(* CoDeSys 2.3.9.41 project: PLC1.pro *)
(* Libraries: Util.lib 18.5.10 15:14:28, STANDARD.LIB 4.10.05 11:14:46, IECSFC.LIB 13.4.06 15:51:28, SYSLIBTIME.LIB 6.11.19 15:29:28, ANALYZATION.LIB 5.10.99 09:05:06 *)

(* PLC configuration (modules and I/O channels)
Fast discrete inputs [I_SIMPLE_INPUT] node 0, in %IB0 out %QB0 {ChannellName = Fast discrete inputs; Filtrationtime = 10000}
  AT %IX0.0 [BitInput] Discrete input 1 {ChannellName = Enter name}
  AT %IX0.1 [BitInput] Discrete input 2 {ChannellName = Enter name}
  AT %IX0.2 [BitInput] Discrete input 3 {ChannellName = Enter name}
  AT %IX0.3 [BitInput] Discrete input 4 {ChannellName = Enter name}
Discrete inputs [ID130] node 1, in %IB1 out %QB1 {ChannellName = Discrete inputs; Filtrationtime_GeneralINP = 10; PinCount = 12; Visibility = No}
  AT %IB1.0 [ByteInput] 8 discrete inputs {ChannellName = Enter name}
  AT %IB1.1 [ByteInput] 4 discrete inputs {ChannellName = Enter name}
DO1 AT %QX2.0 [BitOutput] Fast discrete output 1 {ChannellName = Enter name}
AT %QX2.1 [BitOutput] Fast discrete output 2 {ChannellName = Enter name}
AT %QX2.2 [BitOutput] Fast discrete output 3 {ChannellName = Enter name}
AT %QX2.3 [BitOutput] Fast discrete output 4 {ChannellName = Enter name}
Discrete outputs [ID131] node 3, in %IB3 out %QB3 {ChannellName = Discrete outputs; SafeValueByte = 0; Visibility = No}
  AT %QB3.0 [ByteOutput] 8 discrete outputs {ChannellName = Enter name}
  AT %QB3.1 [ByteOutput] 8 discrete outputs {ChannellName = Enter name}
Fast analog inputs [ID125] node 4, in %IB4 out %QB4 {ChannellName = Fast analog inputs; Flt_Comm = 50Hz 2Por}
  AT %IR4.0 [FloatInputP] You need to reboot PLC after change AI configuration! {ChannellName = Fast analog input; AIN_TYPE = 4-20 mA; Peak_Filtr = 200; Flt_Ch = Off; TauRC = 10; MinFV = 0; MaxFV = 20000.0}
  AT %IR4.1 [FloatInputP] You need to reboot PLC after change AI configuration! {ChannellName = Fast analog input; AIN_TYPE = 4-20 mA; Peak_Filtr = 200; Flt_Ch = Off; TauRC = 10; MinFV = 0; MaxFV = 20000.0}
  AT %IR4.2 [FloatInputP] You need to reboot PLC after change AI configuration! {ChannellName = Fast analog input; AIN_TYPE = 4-20 mA; Peak_Filtr = 200; Flt_Ch = Off; TauRC = 10; MinFV = 0; MaxFV = 20000.0}
  AT %IR4.3 [FloatInputP] You need to reboot PLC after change AI configuration! {ChannellName = Fast analog input; AIN_TYPE = 4-20 mA; Peak_Filtr = 200; Flt_Ch = Off; TauRC = 10; MinFV = 0; MaxFV = 20000.0}
  AT %IR4.4 [FloatInputP] You need to reboot PLC after change AI configuration! {ChannellName = Fast analog input; AIN_TYPE = 4-20 mA; Peak_Filtr = 200; Flt_Ch = Off; TauRC = 10; MinFV = 0; MaxFV = 20000.0}
  AT %IR4.5 [FloatInputP] You need to reboot PLC after change AI configuration! {ChannellName = Fast analog input; AIN_TYPE = 4-20 mA; Peak_Filtr = 200; Flt_Ch = Off; TauRC = 10; MinFV = 0; MaxFV = 20000.0}
  AT %IR4.6 [FloatInputP] You need to reboot PLC after change AI configuration! {ChannellName = Fast analog input; AIN_TYPE = 4-20 mA; Peak_Filtr = 200; Flt_Ch = Off; TauRC = 10; MinFV = 0; MaxFV = 20000.0}
  AT %IR4.7 [FloatInputP] You need to reboot PLC after change AI configuration! {ChannellName = Fast analog input; AIN_TYPE = 4-20 mA; Peak_Filtr = 200; Flt_Ch = Off; TauRC = 10; MinFV = 0; MaxFV = 20000.0}
  AT %IW4.8 [WordInput] AI read time (10ms) {ChannellName = Enter name}
Analog outputs [ID126] node 5, in %IB5 out %QB5 {ChannellName = Analog outputs}
  AT %QR5.0 [FloatOutputP] AO #1 {ChannellName = Analog output; AOUT_TYPE = 4-20 mA; SafeValueREAL = 0.0}
  AT %QR5.1 [FloatOutputP] AO #2 {ChannellName = Analog output; AOUT_TYPE = 4-20 mA; SafeValueREAL = 0.0}
  AT %QR5.2 [FloatOutputP] AO #3 {ChannellName = Analog output; AOUT_TYPE = 4-20 mA; SafeValueREAL = 0.0}
  AT %QR5.3 [FloatOutputP] AO #4 {ChannellName = Analog output; AOUT_TYPE = 4-20 mA; SafeValueREAL = 0.0}
Special input [ID103] node 6, in %IB6 out %QB6 {ChannellName = Special input}
  AT %IX6.0 [BitInput] Special input {ChannellName = Enter name}
Special output [ID104] node 7, in %IB7 out %QB7 {ChannellName = Special output}
  AT %QX7.0 [BitOutput] Special output {ChannellName = Enter name}
ModBus (slave) [MODBUS_ID400] node 8, in %IB8 out %QB8 {ChannellName = ModBus (slave); SlaveIdentificator = 1; Visibility = No}
Debug RS-232 [DEBUG_USART] node 0, in %IB8.0.0 out %QB8.0.0 {ChannellName = Debug RS-232; CommunicationSpeed = 115200; Parity = NO PARITY CHECK; BitLength = 8 bits; StopLength = One stop bit; InterfaceType = RS232; FrameOriented = RTU; Timeout = 0; Visibility = No}
MODBUS_ID400Parameter.ChannellName1Modu AT %QW8.1.0 [WordOutput] e.Register2 byte2 byteSTRING2 byteIB%QB%MB%MTwoByte {ChannellName = Enter name}
AT %QD9.0 [DWordOutput] Last address {ChannellName = Enter name}
AT %QW9.1 [WordOutput] Last error {ChannellName = Enter name}
Empty [Empty_module] node 0, in %IB9.0 out %QB9.0 {ChannellName = Empty slot}
AT %QB9.1.0 [ComChannel] Command (0xff - Start) {ChannellName = Enter name}
read_float_from_PLC2 AT %QD9.1.0.0 [FloatOutput] {ChannellName = Enter name}
uint_to_plc2 AT %QW9.1.1.0 [WordOutput] {ChannellName = Enter name}
AT %QB9.2.0 [ComChannel] Command (0xff - Start) {ChannellName = Enter name}
real_to_pan AT %QD9.2.0.0 [FloatOutput] {ChannellName = Enter name}
uint_from_pan AT %QW9.2.1.0 [WordOutput] {ChannellName = Enter name}
*)

(* POU PLC_PRG, CFC *)
PROGRAM PLC_PRG
VAR
	blinker: BLINK;
	TP: TP;
	boolstub1: BOOL;
	boolstub2: BOOL;
END_VAR
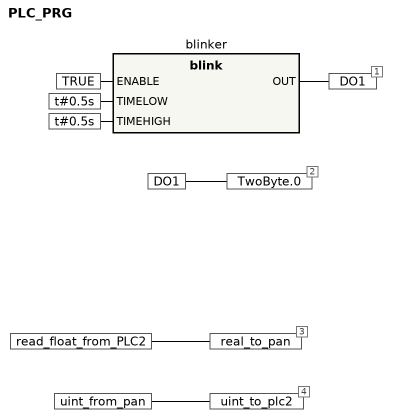
_CFC_ (* Continuous Function Chart, elements in execution order *)
#0 blinker:blink(ENABLE: TRUE, TIMELOW: t#0.5s, TIMEHIGH: t#0.5s)
#1 DO1 <= #0.OUT
#2 TwoByte.0 <= DO1
#3 real_to_pan <= read_float_from_PLC2
#4 uint_to_plc2 <= uint_from_pan
_END_CFC_
(* the same logic as Structured Text *)
blinker(ENABLE := TRUE, TIMELOW := t#0.5s, TIMEHIGH := t#0.5s);
DO1 := blinker.OUT;
TwoByte.0 := DO1;
real_to_pan := read_float_from_PLC2;
uint_to_plc2 := uint_from_pan;
END_PROGRAM
